FUNCTION_BLOCK FbMode
VAR_INPUT
	xAutoModePB: BOOL;
	xManModePB: BOOL;
END_VAR
VAR_OUTPUT
	xAutoMode: BOOL;
	xManMode: BOOL;
END_VAR

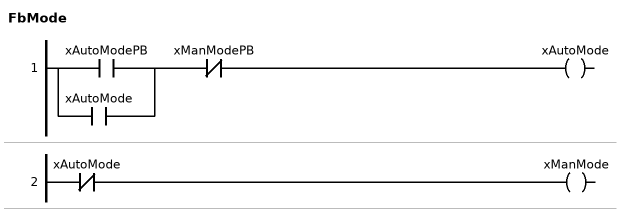
// NETWORK 1
xAutoMode := (xAutoModePB OR xAutoMode) AND NOT xManModePB;

// NETWORK 2
xManMode := NOT xAutoMode;

END_FUNCTION_BLOCK

(* stored: Version 1.1.0.1, ProductVersion 3.1.4024.12
   POU FbMode: Id {a222425f-2260-4292-9171-33dbd345df27}, SpecialFunc None *)
